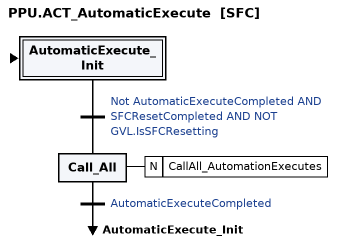
(* [picture p48: PPU.ACT_AutomaticExecute, SFC] *)
INITIAL_STEP AutomaticExecute_Init:
END_STEP
TRANSITION FROM AutomaticExecute_Init TO Call_All
  := Not AutomaticExecuteCompleted AND SFCResetCompleted AND NOT GVL.IsSFCResetting;
END_TRANSITION
STEP Call_All:
  CallAll_AutomationExecutes(N);
END_STEP
TRANSITION FROM Call_All TO AutomaticExecute_Init
  := AutomaticExecuteCompleted;
END_TRANSITION
END_ACTION

ACTION ACT_EmergencyStop:
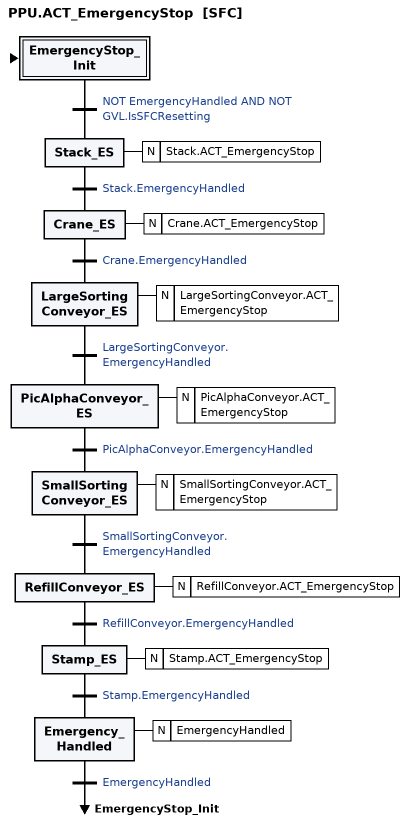
INITIAL_STEP EmergencyStop_Init:
END_STEP
TRANSITION FROM EmergencyStop_Init TO Stack_ES
  := NOT EmergencyHandled AND NOT GVL.IsSFCResetting;
END_TRANSITION
STEP Stack_ES:
  Stack.ACT_EmergencyStop(N);
END_STEP
TRANSITION FROM Stack_ES TO Crane_ES
  := Stack.EmergencyHandled;
END_TRANSITION
STEP Crane_ES:
  Crane.ACT_EmergencyStop(N);
END_STEP
TRANSITION FROM Crane_ES TO LargeSortingConveyor_ES
  := Crane.EmergencyHandled;
END_TRANSITION
STEP LargeSortingConveyor_ES:
  LargeSortingConveyor.ACT_EmergencyStop(N);
END_STEP
TRANSITION FROM LargeSortingConveyor_ES TO PicAlphaConveyor_ES
  := LargeSortingConveyor.EmergencyHandled;
END_TRANSITION
STEP PicAlphaConveyor_ES:
  PicAlphaConveyor.ACT_EmergencyStop(N);
END_STEP
TRANSITION FROM PicAlphaConveyor_ES TO SmallSortingConveyor_ES
  := PicAlphaConveyor.EmergencyHandled;
END_TRANSITION
STEP SmallSortingConveyor_ES:
  SmallSortingConveyor.ACT_EmergencyStop(N);
END_STEP
TRANSITION FROM SmallSortingConveyor_ES TO RefillConveyor_ES
  := SmallSortingConveyor.EmergencyHandled;
END_TRANSITION
STEP RefillConveyor_ES:
  RefillConveyor.ACT_EmergencyStop(N);
END_STEP
TRANSITION FROM RefillConveyor_ES TO Stamp_ES
  := RefillConveyor.EmergencyHandled;
END_TRANSITION
STEP Stamp_ES:
  Stamp.ACT_EmergencyStop(N);
END_STEP
TRANSITION FROM Stamp_ES TO Emergency_Handled
  := Stamp.EmergencyHandled;
END_TRANSITION
STEP Emergency_Handled:
  EmergencyHandled(N);
END_STEP
TRANSITION FROM Emergency_Handled TO EmergencyStop_Init
  := EmergencyHandled;
END_TRANSITION
END_ACTION

ACTION ACT_Init:
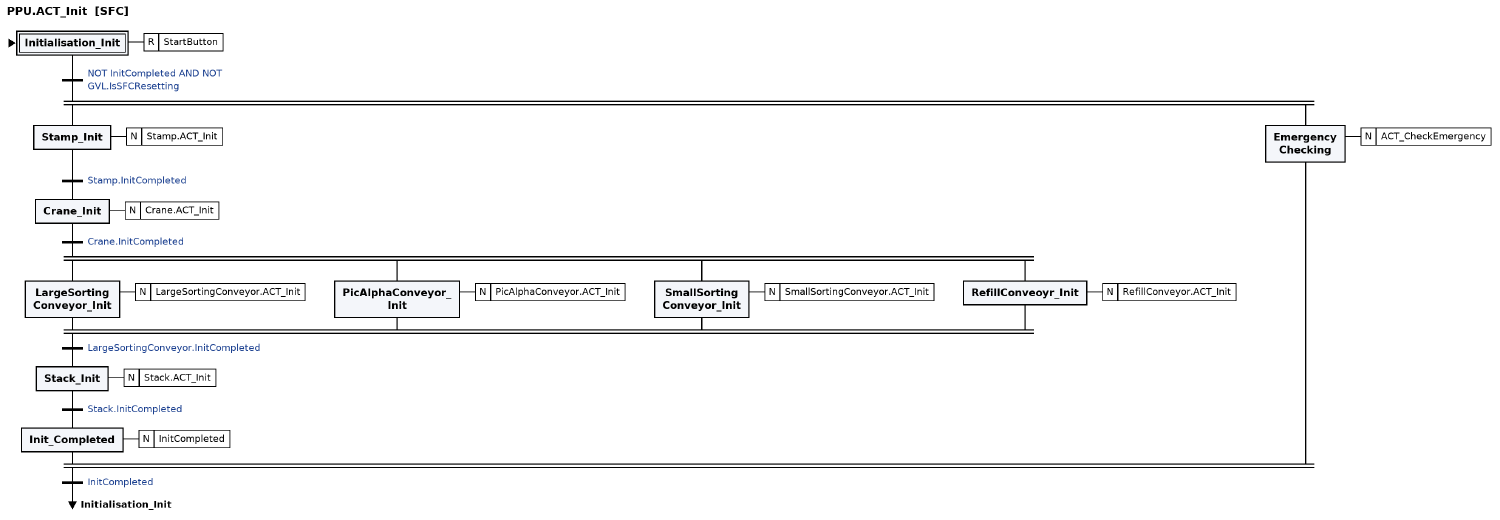
INITIAL_STEP Initialisation_Init:
  StartButton(R);
END_STEP
TRANSITION FROM Initialisation_Init TO (Stamp_Init, EmergencyChecking)
  := NOT InitCompleted AND NOT GVL.IsSFCResetting;
END_TRANSITION
STEP Stamp_Init:
  Stamp.ACT_Init(N);
END_STEP
TRANSITION FROM Stamp_Init TO Crane_Init
  := Stamp.InitCompleted;
END_TRANSITION
STEP Crane_Init:
  Crane.ACT_Init(N);
END_STEP
TRANSITION FROM Crane_Init TO (LargeSortingConveyor_Init, PicAlphaConveyor_Init, SmallSortingConveyor_Init, RefillConveoyr_Init)
  := Crane.InitCompleted;
END_TRANSITION
STEP LargeSortingConveyor_Init:
  LargeSortingConveyor.ACT_Init(N);
END_STEP
TRANSITION FROM (LargeSortingConveyor_Init, PicAlphaConveyor_Init, SmallSortingConveyor_Init, RefillConveoyr_Init) TO Stack_Init
  := LargeSortingConveyor.InitCompleted;
END_TRANSITION
STEP PicAlphaConveyor_Init:
  PicAlphaConveyor.ACT_Init(N);
END_STEP
STEP SmallSortingConveyor_Init:
  SmallSortingConveyor.ACT_Init(N);
END_STEP
STEP RefillConveoyr_Init:
  RefillConveyor.ACT_Init(N);
END_STEP
STEP Stack_Init:
  Stack.ACT_Init(N);
END_STEP
TRANSITION FROM Stack_Init TO Init_Completed
  := Stack.InitCompleted;
END_TRANSITION
STEP Init_Completed:
  InitCompleted(N);
END_STEP
TRANSITION FROM (Init_Completed, EmergencyChecking) TO Initialisation_Init
  := InitCompleted;
END_TRANSITION
STEP EmergencyChecking:
  ACT_CheckEmergency(N);
END_STEP
END_ACTION
END_FUNCTION_BLOCK

CONFIGURATION Application
  RESOURCE Scenario_15 ON PLC
(* global variable list GVL *)
{attribute 'qualified_only'}
VAR_GLOBAL
	IsSFCResetting : BOOL;
END_VAR
    TASK PlcTask(INTERVAL := T#0ms, PRIORITY := 20);
    PROGRAM MAIN WITH PlcTask : MAIN;
  END_RESOURCE
END_CONFIGURATION
